// TIA Portal V20 export
VAR_GLOBAL   // PLC tag table "PROFIsafe Drives"
   BA030AZARDR1_Status AT %I5100.0 : "safety.LDrvSafe_typeSinaTlg901Status";
   BA030AZARDR1_Control AT %Q5100.0 : "safety.LDrvSafe_typeSinaTlg901Control";
   BA030AZARDR2_Status AT %I5140.0 : "safety.LDrvSafe_typeSinaTlg901Status";
   BA030AZARDR2_Control AT %Q5140.0 : "safety.LDrvSafe_typeSinaTlg901Control";
   BA030AZARDR3_Status AT %I5180.0 : "safety.LDrvSafe_typeSinaTlg901Status";
   BA030AZARDR3_Control AT %Q5180.0 : "safety.LDrvSafe_typeSinaTlg901Control";
   BA030AZARDR4_Status AT %I5220.0 : "safety.LDrvSafe_typeSinaTlg901Status";
   BA030AZARDR4_Control AT %Q5220.0 : "safety.LDrvSafe_typeSinaTlg901Control";
   BA030AZARDR5_Status AT %I5254.0 : "safety.LDrvSafe_typeSinaTlg901Status";
   BA030AZARDR5_Control AT %Q5254.0 : "safety.LDrvSafe_typeSinaTlg901Control";
   BA030AZARDR6_Status AT %I5288.0 : "safety.LDrvSafe_typeSinaTlg901Status";
   BA030AZARDR6_Control AT %Q5288.0 : "safety.LDrvSafe_typeSinaTlg901Control";
   BA030AZARDR7_Status AT %I5322.0 : "safety.LDrvSafe_typeSinaTlg901Status";
   BA030AZARDR7_Control AT %Q5322.0 : "safety.LDrvSafe_typeSinaTlg901Control";
   BA030AZARDR8_Status AT %I5356.0 : "safety.LDrvSafe_typeSinaTlg901Status";
   BA030AZARDR8_Control AT %Q5356.0 : "safety.LDrvSafe_typeSinaTlg901Control";
   BA030AZARDR9_Status AT %I5390.0 : "safety.LDrvSafe_typeSinaTlg901Status";
   BA030AZARDR9_Control AT %Q5390.0 : "safety.LDrvSafe_typeSinaTlg901Control";
   BA030AZARDR10_Status AT %I5424.0 : "safety.LDrvSafe_typeSinaTlg901Status";
   BA030AZARDR10_Control AT %Q5424.0 : "safety.LDrvSafe_typeSinaTlg901Control";
   BA030AZARDR11_Status AT %I5468.0 : "safety.LDrvSafe_typeSinaTlg901Status";
   BA030AZARDR11_Control AT %Q5468.0 : "safety.LDrvSafe_typeSinaTlg901Control";
   BA030AZARDR12_Status AT %I5502.0 : "safety.LDrvSafe_typeSinaTlg901Status";
   BA030AZARDR12_Control AT %Q5502.0 : "safety.LDrvSafe_typeSinaTlg901Control";
   BA030AZARDR13_Status AT %I5546.0 : "safety.LDrvSafe_typeSinaTlg901Status";
   BA030AZARDR13_Control AT %Q5546.0 : "safety.LDrvSafe_typeSinaTlg901Control";
   BA030AZARDR14_Status AT %I5590.0 : "safety.LDrvSafe_typeSinaTlg901Status";
   BA030AZARDR14_Control AT %Q5590.0 : "safety.LDrvSafe_typeSinaTlg901Control";
   BA030AZARDR15_Status AT %I5634.0 : "safety.LDrvSafe_typeSinaTlg901Status";
   BA030AZARDR15_Control AT %Q5634.0 : "safety.LDrvSafe_typeSinaTlg901Control";
   BA030AZARDR16_Status AT %I5668.0 : "safety.LDrvSafe_typeSinaTlg901Status";
   BA030AZARDR16_Control AT %Q5668.0 : "safety.LDrvSafe_typeSinaTlg901Control";
   BA030AZARDR17_Status AT %I5702.0 : "safety.LDrvSafe_typeSinaTlg901Status";
   BA030AZARDR17_Control AT %Q5702.0 : "safety.LDrvSafe_typeSinaTlg901Control";
   BA030AZARDR18_Status AT %I5736.0 : "safety.LDrvSafe_typeSinaTlg901Status";
   BA030AZARDR18_Control AT %Q5736.0 : "safety.LDrvSafe_typeSinaTlg901Control";
   BA030AZARDR19_Status AT %I5770.0 : "safety.LDrvSafe_typeSinaTlg901Status";
   BA030AZARDR19_Control AT %Q5770.0 : "safety.LDrvSafe_typeSinaTlg901Control";
   BA030AZARDR20_Status AT %I5804.0 : "safety.LDrvSafe_typeSinaTlg901Status";
   BA030AZARDR20_Control AT %Q5804.0 : "safety.LDrvSafe_typeSinaTlg901Control";
   BA030AZARDR21_Status AT %I5838.0 : "safety.LDrvSafe_typeSinaTlg901Status";
   BA030AZARDR21_Control AT %Q5838.0 : "safety.LDrvSafe_typeSinaTlg901Control";
   BA030AZARDR22_Status AT %I5872.0 : "safety.LDrvSafe_typeSinaTlg901Status";
   BA030AZARDR22_Control AT %Q5872.0 : "safety.LDrvSafe_typeSinaTlg901Control";
   BA030AZARDR23_Status AT %I5906.0 : "safety.LDrvSafe_typeSinaTlg901Status";
   BA030AZARDR23_Control AT %Q5906.0 : "safety.LDrvSafe_typeSinaTlg901Control";
   BA030AZARDR24_Status AT %I5940.0 : "safety.LDrvSafe_typeSinaTlg901Status";
   BA030AZARDR24_Control AT %Q5940.0 : "safety.LDrvSafe_typeSinaTlg901Control";
   BA030AZARDR25_Status AT %I5984.0 : "safety.LDrvSafe_typeSinaTlg901Status";
   BA030AZARDR25_Control AT %Q5984.0 : "safety.LDrvSafe_typeSinaTlg901Control";
   BA030AZARDR26_Status AT %I6018.0 : "safety.LDrvSafe_typeSinaTlg901Status";
   BA030AZARDR26_Control AT %Q6018.0 : "safety.LDrvSafe_typeSinaTlg901Control";
   BA030AZARDR27_Status AT %I6062.0 : "safety.LDrvSafe_typeSinaTlg901Status";
   BA030AZARDR27_Control AT %Q6062.0 : "safety.LDrvSafe_typeSinaTlg901Control";
   BA030AZARDR28_Status AT %I6096.0 : "safety.LDrvSafe_typeSinaTlg901Status";
   BA030AZARDR28_Control AT %Q6096.0 : "safety.LDrvSafe_typeSinaTlg901Control";
   BA030AZARDR29_Status AT %I6140.0 : "safety.LDrvSafe_typeSinaTlg901Status";
   BA030AZARDR29_Control AT %Q6140.0 : "safety.LDrvSafe_typeSinaTlg901Control";
   BA030AZARDR30_Status AT %I6174.0 : "safety.LDrvSafe_typeSinaTlg901Status";
   BA030AZARDR30_Control AT %Q6174.0 : "safety.LDrvSafe_typeSinaTlg901Control";
   BA030AZARDR31_Status AT %I6218.0 : "safety.LDrvSafe_typeSinaTlg901Status";
   BA030AZARDR31_Control AT %Q6218.0 : "safety.LDrvSafe_typeSinaTlg901Control";
   BA030AZARDR32_Status AT %I6262.0 : "safety.LDrvSafe_typeSinaTlg901Status";
   BA030AZARDR32_Control AT %Q6262.0 : "safety.LDrvSafe_typeSinaTlg901Control";
   BA030AZARDR33_Status AT %I6306.0 : "safety.LDrvSafe_typeSinaTlg901Status";
   BA030AZARDR33_Control AT %Q6306.0 : "safety.LDrvSafe_typeSinaTlg901Control";
   BA030AZARDR34_Status AT %I6350.0 : "safety.LDrvSafe_typeSinaTlg901Status";
   BA030AZARDR34_Control AT %Q6350.0 : "safety.LDrvSafe_typeSinaTlg901Control";
   BA030AZARDR35_Status AT %I6384.0 : "safety.LDrvSafe_typeSinaTlg901Status";
   BA030AZARDR35_Control AT %Q6384.0 : "safety.LDrvSafe_typeSinaTlg901Control";
   BA030AZARDR36_Status AT %I6428.0 : "safety.LDrvSafe_typeSinaTlg901Status";
   BA030AZARDR36_Control AT %Q6428.0 : "safety.LDrvSafe_typeSinaTlg901Control";
   BA030AZARDR37_Status AT %I6462.0 : "safety.LDrvSafe_typeSinaTlg901Status";
   BA030AZARDR37_Control AT %Q6462.0 : "safety.LDrvSafe_typeSinaTlg901Control";
   BA030AZARDR38_Status AT %I6506.0 : "safety.LDrvSafe_typeSinaTlg901Status";
   BA030AZARDR38_Control AT %Q6506.0 : "safety.LDrvSafe_typeSinaTlg901Control";
   BA030AZARDR39_Status AT %I6540.0 : "safety.LDrvSafe_typeSinaTlg901Status";
   BA030AZARDR39_Control AT %Q6540.0 : "safety.LDrvSafe_typeSinaTlg901Control";
   BA030AZARDR40_Status AT %I6574.0 : "safety.LDrvSafe_typeSinaTlg901Status";
   BA030AZARDR40_Control AT %Q6574.0 : "safety.LDrvSafe_typeSinaTlg901Control";
   BA030AZARDR41_Status AT %I6608.0 : "safety.LDrvSafe_typeSinaTlg901Status";
   BA030AZARDR41_Control AT %Q6608.0 : "safety.LDrvSafe_typeSinaTlg901Control";
END_VAR
